FUNCTION_BLOCK FB_Camera
VAR_INPUT
END_VAR
VAR_OUTPUT
END_VAR
VAR
	Trigger	AT %Q*			: BOOL;				// signal to take picture and analyze
	CameraData				: ST_CameraData;	// modbus camera data
	VisionStatus			: ARRAY[0..3] OF BYTE;// modbus camera status
	_tubeParameters			: ST_TubeParameters;
	_pass					: BOOL;
	_fail					: BOOL;
	_noDetect				: BOOL;
			
	_xPoints 				: ARRAY[1..GVL.NumberVisionPoints] OF LREAL;
	_yPoints 				: ARRAY[1..GVL.NumberVisionPoints] OF LREAL;
	_xEllipsePoints			: ARRAY[1..GVL.NumberEllipsePoints] OF LREAL;
	_yEllipsePoints			: ARRAY[1..GVL.NumberEllipsePoints] OF LREAL;
		
	_displayVisionPts		: ARRAY[1..2,1..GVL.NumberVisionPoints] OF LREAL;
	_displayEllipsePts		: ARRAY[1..2,1..GVL.NumberEllipsePoints] OF LREAL;
	_columnPeak				: LREAL;	// xPeak value of the vision points
	_rowPeak				: LREAL;	// yPeak value of the vision points
	_rowCenterLine			: LREAL;	// based on entered minor value -> y value at the center-line axis
	_minorCalculated 		: LREAL;
	_majorCalculated		: LREAL;
	_xEllipseCenter			: LREAL;
	_yEllipseCenter			: LREAL;

	(* for calculating the pitch *)	
	_patternX1				: LREAL;
	_patternX2				: LREAL;
	_patternX3				: LREAL;
	_patternY1				: LREAL;
	_patternY2				: LREAL;
	_patternY3				: LREAL;
	
	(* calculation variables *)
	DeltaXpx				: LREAL;	// distance from peak of curve to center of cut (row)
	DeltaYpx				: LREAL;	// distance from peak of curve to center of cut (column)
	CutLength				: LREAL;
	CutHeight				: LREAL;
	DeltaXmm				: LREAL;
	DeltaYmm				: LREAL;
	(* results *)
	_CutLengthWithOffset	: LREAL;
	_DeltaXmmWithOffset		: LREAL;
	_DeltaYmmWithOffset		: LREAL;
	
	_depthOffset			: REAL; 				// difference due to the plane of cut is different than plane of pattern detect
	_minorRadiusMm			: LREAL := 2.5955;		// minor radius of ellipse in mm
	_majorRadiusMm			: LREAL;
	_slitCenterApparentRow	: LREAL;				// [px] this is the center of the part in x when accounting for the offset due to vision plane versus cut plane
	_tubeCenter				: LREAL;
	_tubeCenterOffset		: LREAL;
	_tubeCenterWithOffset	: LREAL;
	_cameraProgram			: STRING;
	_previousTubeIndex		: INT;
	
	_hmiParameters			: ST_CameraParameters;
	_parameters				: ST_CameraParameters;
	fbMessageChange			: FB_TcMessage;
	fbMessageLoaded			: FB_TcMessage;
END_VAR

PROPERTY angle : LREAL
GET
angle := _parameters.angle;
END_GET
SET
fbMessageChange.ipArguments.Clear().AddString('Angle').AddLReal(_parameters.angle).AddLReal(angle);
fbMessageChange.Send(0);
_parameters.angle := angle;
END_SET
END_PROPERTY

METHOD Calibrate : BOOL
VAR_INPUT
END_VAR
_hmiParameters.pitchRow := (CalibrationDistance / ABS(PatternY1 - PatternY2));
_hmiParameters.pitchColumn := (CalibrationDistance / ABS(PatternX2 - PatternX3));
END_METHOD

PROPERTY CalibrationDistance : LREAL
GET
CalibrationDistance := _parameters.calibrationDistance;
END_GET
SET
fbMessageChange.ipArguments.Clear().AddString('Calibration Distance').AddLReal(_parameters.calibrationDistance).AddLReal(CalibrationDistance);
fbMessageChange.Send(0);
_parameters.calibrationDistance := CalibrationDistance;
END_SET
END_PROPERTY

PROPERTY CameraProgram : STRING
GET
CameraProgram := _cameraProgram;
END_GET
SET
_cameraProgram := CameraProgram;
END_SET
END_PROPERTY

METHOD Compute : INT
VAR_INPUT
	Execute		: BOOL;
END_VAR
VAR_INST
	rTrig			: R_TRIG;
	nIndex			: INT;
	fbSecond		: FB_SecondOrder;
 	fbFourth		: FB_FourthOrder;
	fbEllipse		: FB_Ellipse;
	zeroValues		: BOOL;
END_VAR

VAR
	i: INT;
	yValue	: LREAL;
END_VAR
(* when computing the new cut positions, subtract the delta values from the 
original cut positions *)

rTrig(CLK := Execute);
IF rTrig.Q THEN
	nIndex := 10;
END_IF

IF NOT Execute THEN
	nIndex := 0;
END_IF

CASE nIndex OF
	0: // idle state
		Compute := 0;
	10: // get data
		IF GetCameraData() = 1 THEN
			nIndex := 15;
		END_IF
	15: // did pattern match find _xPoints, _yPoints?
		zeroValues := FALSE;
		FOR i := 1 TO GVL.NumberVisionPoints DO
			IF _xPoints[i] = 0 OR _yPoints[i] = 0 THEN
				zeroValues := TRUE;
			END_IF
		END_FOR
		IF zeroValues THEN
			nIndex := 60;
		ELSE
			nIndex := 20;
		END_IF
	20: // compute the peak x value of the data		
		fbSecond.FindPeak(xValues := ADR(_xPoints), yValues := ADR(_yPoints), xPeak := ADR(_columnPeak));
		fbFourth.FindYatX(xValues := ADR(_xPoints), yValues := ADR(_yPoints), xPeak := ADR(_columnPeak), yPeak := ADR(_rowPeak));
		DeltaYpx := CameraData.Results.LocationInX - _columnPeak;
		DeltaYmm := DeltaYpx * _hmiParameters.pitchColumn;
		_DeltaYmmWithOffset := DeltaYmm + _tubeParameters.AdjustmentY;
		
		CutLength := CameraData.Results.WidthMeasurement * _hmiParameters.pitchColumn;		
		_CutLengthWithOffset := CutLength + _tubeParameters.AdjustmentLength;
		CutHeight := CameraData.Results.HeightMeasurement * _hmiParameters.pitchRow;
		
		_tubeCenter := _rowPeak + 0.5*_tubeParameters.Diameter /_hmiParameters.pitchRow;
		_tubeCenterOffset := (_tubeParameters.DepthOfPocket*TAN(_hmiParameters.angle * 2*3.14159/360.0))/_hmiParameters.pitchRow;
		_tubeCenterWithOffset := _tubeCenter + _tubeCenterOffset;
		
		DeltaXpx := (CameraData.Results.LocationInY - 0.5*CameraData.Results.HeightMeasurement) - _tubeCenterWithOffset;
		DeltaXmm := DeltaXpx * _hmiParameters.pitchRow;
		_DeltaXmmWithOffset := DeltaXmm + _tubeParameters.AdjustmentX;
		
		nIndex := 50;
	30: // compute ellipse
		fbEllipse.EllipseFit(xValues := _xEllipsePoints, yValues := _yEllipsePoints);
		nIndex := 40;
		
	40: // assign values
		_minorCalculated := fbEllipse.minor;
		_majorCalculated := fbEllipse.major;
		_xEllipseCenter := fbEllipse.centrex;
		_yEllipseCenter := fbEllipse.centrey;
		nIndex := 50;
	50: // done state
		Compute := 1;		
	60: // didn't find the pattern, so can't compute a peak
		Compute := -1;					
END_CASE
END_METHOD

PROPERTY CutLengthWithOffset : LREAL
GET
CutLengthWithOffset := _CutLengthWithOffset;
END_GET
END_PROPERTY

PROPERTY DeltaXmmWithOffset : LREAL
GET
DeltaXmmWithOffset := _DeltaXmmWithOffset;
END_GET
END_PROPERTY

PROPERTY DeltaYmmWithOffset : LREAL
GET
DeltaYmmWithOffset := _DeltaYmmWithOffset;
END_GET
END_PROPERTY

PROPERTY Fail : BOOL
GET
Fail := _fail;
END_GET
SET
_fail := Fail;
END_SET
END_PROPERTY

METHOD FB_init : BOOL
VAR_INPUT
	bInitRetains : BOOL; // if TRUE, the retain variables are initialized (warm start / cold start)
	bInCopyCode : BOOL;  // if TRUE, the instance afterwards gets moved into the copy code (online change)
END_VAR
IF NOT fbMessageChange.EqualsToEventEntryEx(stOther := TC_EVENTS.SlitterEvents.ParameterChange) THEN
	fbMessageChange.CreateEx(TC_EVENTS.SlitterEvents.ParameterChange, 0);
	fbMessageChange.ipArguments.Clear();
END_IF

IF NOT fbMessageLoaded.EqualsToEventEntryEx(stOther := TC_EVENTS.SlitterEvents.ParametersLoadedFromFile) THEN
	fbMessageLoaded.CreateEx(TC_EVENTS.SlitterEvents.ParametersLoadedFromFile, 0);
	fbMessageLoaded.ipArguments.Clear().AddString('Camera');
END_IF
END_METHOD

METHOD GetCameraData : INT
VAR_INPUT
END_VAR

VAR_INST
	i				: INT;
	fbMBRegRead		: FB_MBReadRegs;
END_VAR
// format on Cognex needs to be little endian 
GetCameraData := 0;
fbMBRegRead.bExecute := TRUE;

fbMBRegRead.sIPAddr := GVL.CameraIpAddress;
fbMBRegRead.nTCPPort := 502;
fbMBRegRead.nUnitID := 16#FF;
fbMBRegRead.nQuantity := 94; // 188/2;
fbMBRegRead.nMBAddr := GVL.ModbusReadOffset+5;
fbMBRegRead.cbLength := SIZEOF(CameraData.Results);
fbMBRegRead.pDestAddr := ADR(CameraData.Results);

fbMBRegRead();

IF NOT fbMBRegRead.bBusy THEN
	IF NOT fbMBRegRead.bError THEN
		fbMBRegRead(bExecute := FALSE);
		FOR i := 1 TO GVL.NumberVisionPoints DO
			_yPoints[i] := REAL_TO_LREAL(CameraData.Results.PointValueRow[i]);
			_xPoints[i] := REAL_TO_LREAL(CameraData.Results.PointValueColumn[i]);
			_displayVisionPts[1,i] := INT_TO_LREAL(LREAL_TO_INT(_xPoints[i]*100))/100.0; // column values
			_displayVisionPts[2,i] := INT_TO_LREAL(LREAL_TO_INT(_yPoints[i]*100))/100.0; // row values	
		END_FOR

		GetCameraData := 1;	
	ELSE
		fbMBRegRead(bExecute := FALSE);
		FOR i := 1 TO GVL.NumberVisionPoints DO
			_xPoints[i] := 0;
			_yPoints[i] := 0;
			_displayVisionPts[1,i] := 0;
			_displayVisionPts[2,i] := 0;
	
		END_FOR
		GetCameraData := -1;	
		
	END_IF
END_IF
END_METHOD

METHOD Inspect : INT
VAR_INPUT
	Execute	: BOOL;
END_VAR
VAR_INST
	nIndex 	: INT;
	rTrig	: R_TRIG;
	CountStart : REAL;
	CountFinish : REAL;
	Count	: REAL;
	CameraTON	: TON := (PT := T#250MS);
	CameraDataResult : INT;
END_VAR
rTrig(CLK := Execute);
IF rTrig.Q THEN
	Inspect := 0;
	nIndex := 10;
	Trigger := FALSE;
	Compute(Execute := FALSE);
	CameraTON(IN := FALSE);
END_IF

IF NOT Execute THEN
	nIndex := 0;
END_IF

CASE nIndex OF
	0: // idle state
		Inspect := 0;
	10: // trigger the camera
		IF GetCameraData() = 1 THEN
			Count := CameraData.Results.Count;
			CountStart := CameraData.Results.Count;
			nIndex := 11;
		END_IF
	11: // trigger camera
		Trigger := TRUE;
		nIndex := 12;
	12: // wait 250 ms
		CameraTON.IN := TRUE;
		IF CameraTON.Q THEN
			CameraTON.IN := FALSE;
			nIndex := 15;
		END_IF
		CameraTON();
	15: // wait for data to be updated
		CameraDataResult := GetCameraData();
		IF CameraDataResult = 1 THEN
			IF Count <> CameraData.Results.Count THEN
				CountFinish := CameraData.Results.Count;
				nIndex := 20;
				Trigger := FALSE;
			END_IF
		END_IF
	20: // Gather the data and analyze locations, etc.
		CameraDataResult := Compute(Execute := TRUE);
		IF CameraDataResult = 1 THEN	// could compute b/c found pattern
			Compute(Execute := FALSE);
			nIndex := 30;	
		ELSIF CameraDataResult = -1 THEN	// could not comput b/c no pattern found
			Compute(Execute := FALSE);
			nIndex := 50;
		END_IF
	30: // compute pass fail
		IF PassFail() THEN	// true = pass
			_pass := TRUE;
			_fail := FALSE;
			_noDetect := FALSE;
		ELSE
			_pass := FALSE;
			_fail := TRUE;
			_noDetect := FALSE;
		END_IF
		nIndex := 40;
	40: // done state
		Inspect := 1;
	50: // error state
		Inspect := -1;
		_noDetect := TRUE;		
		_pass := FALSE;
		_fail := FALSE;		
END_CASE
END_METHOD

METHOD MonitorParameters : BOOL
VAR_INPUT
END_VAR
IF angle <> _hmiParameters.angle THEN
	angle := _hmiParameters.angle;
END_IF

IF CalibrationDistance <> _hmiParameters.calibrationDistance THEN
	CalibrationDistance := _hmiParameters.calibrationDistance;
END_IF

IF pitchColumn <> _hmiParameters.pitchColumn THEN
	pitchColumn := _hmiParameters.pitchColumn;
END_IF

IF pitchRow <> _hmiParameters.pitchRow THEN
	pitchRow := _hmiParameters.pitchRow;
END_IF
END_METHOD

PROPERTY NoDetect : BOOL
GET
NoDetect := _noDetect;
END_GET
SET
_noDetect := NoDetect;
END_SET
END_PROPERTY

PROPERTY Parameters : ST_CameraParameters
GET
Parameters := _parameters;
END_GET
SET
_parameters := Parameters;
_hmiParameters := Parameters;
fbMessageLoaded.Send(0);
END_SET
END_PROPERTY

PROPERTY Pass : BOOL
GET
Pass := _pass;
END_GET
SET
_pass := Pass;
END_SET
END_PROPERTY

METHOD PassFail : BOOL
VAR_INPUT
END_VAR
PassFail := TRUE; // set to pass and overwrite if anything causes failure;

// cut length
IF _tubeParameters.AdjustmentLength + CutLength > _tubeParameters.MaxLength OR
	_tubeParameters.AdjustmentLength + CutLength < _tubeParameters.MinLength THEN
		PassFail := FALSE;
END_IF

// delta x
IF ABS(_tubeParameters.AdjustmentX + DeltaXmm) > _tubeParameters.ResultToleranceX THEN
	PassFail := FALSE;
END_IF

// delta y
IF ABS(_tubeParameters.AdjustmentY + DeltaYmm) > _tubeParameters.ResultToleranceY THEN
	PassFail := FALSE;
END_IF

// height
IF CutHeight < _tubeParameters.MinHeight OR CutHeight > _tubeParameters.MaxHeight THEN
	PassFail := FALSE;
END_IF
END_METHOD

PROPERTY PatternMatchX : LREAL
GET
PatternMatchX := REAL_TO_LREAL(CameraData.Results.PatternMatchColumn);
END_GET
END_PROPERTY

PROPERTY PatternMatchY : LREAL
GET
PatternMatchY := REAL_TO_LREAL(CameraData.Results.PatternMatchRow);
END_GET
END_PROPERTY

PROPERTY PatternX1 : LREAL
GET
PatternX1 := _patternX1;
END_GET
SET
_patternX1 := PatternX1;
END_SET
END_PROPERTY

PROPERTY PatternX2 : LREAL
GET
PatternX2 := _patternX2;
END_GET
SET
_patternX2 := PatternX2;
END_SET
END_PROPERTY

PROPERTY PatternX3 : LREAL
GET
PatternX3 := _patternX3;
END_GET
SET
_patternX3 := PatternX3;
END_SET
END_PROPERTY

PROPERTY PatternY1 : LREAL
GET
PatternY1 := _patternY1;
END_GET
SET
_patternY1 := PatternY1;
END_SET
END_PROPERTY

PROPERTY PatternY2 : LREAL
GET
PatternY2 := _patternY2;
END_GET
SET
_patternY2 := PatternY2;
END_SET
END_PROPERTY

PROPERTY PatternY3 : LREAL
GET
PatternY3 := _patternY3;
END_GET
SET
_patternY3 := PatternY3;
END_SET
END_PROPERTY

PROPERTY pitchColumn : LREAL
GET
pitchColumn := _parameters.pitchColumn;
END_GET
SET
fbMessageChange.ipArguments.Clear().AddString('pitchColumn').AddLReal(_parameters.pitchColumn).AddLReal(pitchColumn);
fbMessageChange.Send(0);
_parameters.pitchColumn := pitchColumn;
END_SET
END_PROPERTY

PROPERTY PitchMmToPixel : LREAL
GET
PitchMmToPixel := _hmiParameters.pitchRow;
END_GET
END_PROPERTY

PROPERTY pitchRow : LREAL
GET
pitchRow := _parameters.pitchRow;
END_GET
SET
fbMessageChange.ipArguments.Clear().AddString('pitchRow').AddLReal(_parameters.pitchRow).AddLReal(pitchRow);
fbMessageChange.Send(0);
_parameters.pitchRow := pitchRow;
END_SET
END_PROPERTY

METHOD SelectCameraProgram : INT
VAR_INPUT
	Execute	: BOOL;
END_VAR
VAR_INST
	fbMBRegWrite 	: FB_MBWriteRegs;	// for writing command, name; offset is 2000
	fbMBCoilWrite	: FB_MBWriteCoils;	// for writing vision control; offset is 0
	fbMBReadInputs 	: FB_MBReadInputs; 	// for reading vision status; offset is 0
	nIndex			: INT;
	rTrig			: R_TRIG;
	JobLoadByName 	: WORD := 16#4000;
	temp 			: UDINT := 0;
	info 			: BOOL;
	i 				: WORD;
	strJobName 		: STRING;
	Message			: STRING(255);
	ErrorId			: UDINT;
	nQuantity 		: WORD;
	cbLength 		: UDINT;	
	attempt			: INT;
	attempt2		: INT;	
END_VAR
VAR
END_VAR
rTrig(CLK := Execute);
IF rTrig.Q THEN
	nIndex := 10;
	Message := '';
	ErrorId := 0;
	Attempt := 0;
	Attempt2 := 0;
	fbMBCoilWrite(
		bExecute := FALSE,
		sIPAddr := GVL.CameraIpAddress,
		nTCPPort := 502,
		nUnitID := 16#FF);
	fbMBRegWrite(
		bExecute := FALSE,
		sIPAddr := GVL.CameraIpAddress,
		nTCPPort := 502,
		nUnitID := 16#FF);
	fbMBReadInputs(
		bExecute := FALSE,
		sIPAddr := GVL.CameraIpAddress,
		nTCPPort := 502,
		nUnitID := 16#FF);
END_IF

IF NOT Execute THEN
	nIndex := 0;
END_IF

CASE nIndex OF
	0: // idle state
		SelectCameraProgram := 0;
	10: // check if the program needs to change
		IF _previousTubeIndex = _tubeParameters.Index THEN
			nIndex := 75;
		ELSE
			nIndex := 15;
		END_IF
	15: // Reset everything to zero
		fbMBCoilWrite(
			nQuantity := 32,
			nMBAddr := 0,
			cbLength := 4,
			pSrcAddr := ADR(temp),
			bExecute := TRUE);
		IF NOT fbMBCoilWrite.bBusy THEN
			fbMBCoilWrite(bExecute := FALSE);
			nIndex := 20;
		END_IF
		IF fbMBCoilWrite.bError THEN
			Message := 'Error in state 15';
			ErrorId := fbMBCoilWrite.nErrId;
			fbMBCoilWrite(bExecute := FALSE);
			nIndex := 85;
		END_IF
	20: // place camera offline by setting the set offline bit high 
		// modbus coil offset is 0
		// byte 0, bit 7 is the bit for forcing the camera to be offline
		info := TRUE;
		fbMBCoilWrite(
			sIPAddr := GVL.CameraIpAddress,
			nTCPPort := 502,
			nUnitID := 16#FF,
			nQuantity := 1,
			nMBAddr := 7,
			cbLength := 1,
			pSrcAddr := ADR(Info),
			bExecute := TRUE);
		IF NOT fbMBCoilWrite.bBusy THEN
			fbMBCoilWrite(bExecute := FALSE);
			nIndex := 30;
			END_IF
		IF fbMBCoilWrite.bError THEN
			Message := 'Error in state 20';
			ErrorId := fbMBCoilWrite.nErrId;
			fbMBCoilWrite(bExecute := FALSE);
			nIndex := 85;
		END_IF		
	30: // write the job load by name command into Word 0 of the input block 
		// job load by name command is 0x4000
		// this goes into holding register start which is at 2000
		fbMBRegWrite(
			nQuantity := 1,
			nMBAddr := GVL.ModbusWriteOffset,
			cbLength := 2,
			pSrcAddr := ADR(JobLoadByName),
			bExecute := TRUE);
		IF NOT fbMBRegWrite.bBusy THEN
			fbMBRegWrite(bExecute := FALSE);
			attempt := attempt + 1;
			IF attempt > 2 THEN
				attempt := 0;
				nIndex := 40;
			END_IF
		END_IF
		IF fbMBRegWrite.bError THEN
			Message := 'Error in state 30';
			ErrorId := fbMBRegWrite.nErrId;
			fbMBRegWrite(bExecute := FALSE);
			nIndex := 85;

		END_IF
	40: // write the job name to Word 1 - 2000 (UserData).  Job name must be null terminated
		// a 0 must be in the byte immediately following the job name
		strJobName := CONCAT('SDCARD/Tube', INT_TO_STRING(_tubeParameters.Index));
		strJobName := CONCAT(strJobName, '.job');
		cbLength := 18; // INT_TO_UDINT(LEN(strJobName) + 1);
		nQuantity := 9; //REAL_TO_WORD(UDINT_TO_REAL(cbLength)/2);
		fbMBRegWrite(
			bExecute := TRUE,
			nQuantity := nQuantity,
			nMBAddr := GVL.ModbusWriteOffset + 1,
	//		nQuantity := nQuantity, // number of words
			cbLength := cbLength, // byte size
			pSrcAddr := ADR(strJobName));
		IF NOT fbMBRegWrite.bBusy THEN
			fbMBRegWrite(bExecute := FALSE);
			nIndex := 50;
		END_IF			
		IF fbMBRegWrite.bError THEN
			Message := 'Error in state 40';
			ErrorId := fbMBRegWrite.nErrId;
			fbMBRegWrite(bExecute := FALSE);
			Attempt2 := Attempt2 + 1;
			IF attempt2 > 2 THEN
				nIndex := 85;
			END_IF
		END_IF
		
	50: // Set the Execute Command bit in the vision control block
		//VisionControl.ExecuteCommand := TRUE;
		// Byte 0, bit 4 of vision control 
		info := TRUE;
		fbMBCoilWrite(
			nQuantity := 1,
			nMBAddr := 4,
			cbLength := 1,
			pSrcAddr := ADR(Info),
			bExecute := TRUE);
		IF NOT fbMBCoilWrite.bBusy THEN
			fbMBCoilWrite(bExecute := FALSE);
			nIndex := 60;
		END_IF
		IF fbMBCoilWrite.bError	THEN
			fbMBCoilWrite(bExecute := FALSE);
			nIndex := 85;
			Message := 'error in state 50';
			errorid := fbMBCoilWrite.nErrId;
		END_IF
	60: // wait for command complete of command failed to be set before clearing the execute
		// command bit and the offline bit
		fbMBReadInputs(
			sIPAddr := GVL.CameraIpAddress,
			nTCPPort := 502,
			nUnitID := 16#FF,
			nQuantity := 32,
			nMBAddr := 0,
			cbLength := 4,
			pDestAddr := ADR(VisionStatus),
			bExecute := TRUE);
		IF NOT fbMBReadInputs.bBusy THEN
			fbMBReadInputs(bExecute := FALSE);
			IF VisionStatus[1].6 OR VisionStatus[1].5 THEN
				nIndex := 70;
				IF VisionStatus[1].6 THEN
					nIndex := 80;
					Message := 'VisionSatus[1].6 is true.';
				END_IF
			END_IF
		END_IF
		IF fbMBReadInputs.bError THEN
			fbMBReadInputs(bExecute := FALSE);
			nIndex := 85;
			Errorid := fbMBReadInputs.nErrId;
			Message := 'errror in state 60.';
		END_IF
	70: // done state
		fbMBCoilWrite(
			nQuantity := 32,
			nMBAddr := 0,
			cbLength := 4,
			pSrcAddr := ADR(temp),
			bExecute := TRUE);
		IF NOT fbMBCoilWrite.bBusy THEN
			fbMBCoilWrite(bExecute := FALSE);
			nIndex := 75;
		END_IF
		IF fbMBCoilWrite.bError THEN
			fbMBCoilWrite(bExecute := FALSE);
			nIndex := 85;
			Message := 'error in state 70';
			ErrorID := fbMBCoilWrite.nErrId;			
		END_IF
	75: // done state
		_previousTubeIndex := _tubeParameters.Index;
		SelectCameraProgram := 1;
	80: // error state
		fbMBCoilWrite(
			nQuantity := 32,
			nMBAddr := 0,
			cbLength := 4,
			pSrcAddr := ADR(temp),
			bExecute := TRUE);
		IF NOT fbMBCoilWrite.bBusy THEN
			fbMBCoilWrite(bExecute := FALSE);
			nIndex := 85;
		END_IF

	85: // error state
		SelectCameraProgram := -1;
END_CASE





(*
SelectCameraProgram := 0;
fbMBRegWrite.bExecute := TRUE;

fbMBRegWrite.sIPAddr := GVL.CameraIpAddress;
fbMBRegWrite.nTCPPort := 502;
fbMBRegWrite.nUnitID := 16#FF;
fbMBRegWrite.nQuantity := 2; // words to write
fbMBRegWrite.nMBAddr := GVL.ModbusWriteOffset;
fbMBRegWrite.cbLength := SIZEOF(_tubeSelection);
fbMBRegWrite.pSrcAddr := ADR(_tubeSelection);

fbMBRegWrite();

IF NOT fbMBRegWrite.bBusy THEN
	IF NOT fbMBRegWrite.bError THEN
		fbMBRegWrite(bExecute := FALSE);
		SelectCameraProgram := 1;
	ELSE
		fbMBRegWrite(bExecute := FALSE);
		SelectCameraProgram := -1;		
	END_IF
END_IF
*)
END_METHOD

METHOD TriggerCamera : BOOL
VAR_INPUT
	Execute	: BOOL;
END_VAR
VAR_INST
	rTrig	: R_TRIG;
	nIndex	: INT;
	Counter	: REAL;
END_VAR
rTrig(CLK := Execute);
IF rTrig.Q THEN
	nIndex := 10;
	Trigger	:= FALSE;
END_IF

IF NOT Execute THEN
	nIndex := 0;
END_IF

CASE nIndex OF
	0: // idle state
		TriggerCamera := FALSE;
	10: // get the camera count
		IF GetCameraData() = 1 THEN
			Counter := CameraData.Results.Count;
			nIndex := 20;
		END_IF
	20: // trigger the camera	
		Trigger := TRUE;
		IF GetCameraData() = 1 THEN
			nIndex := 30;
		END_IF
	30: // updated?
		IF Counter <> CameraData.Results.Count THEN
			Trigger := FALSE;
			nIndex := 40;
		ELSE
			nIndex := 20;
		END_IF
	40: // done state
		TriggerCamera := TRUE;
END_CASE
END_METHOD

PROPERTY TubeParameters : ST_TubeParameters
GET
TubeParameters := _tubeParameters;
END_GET
SET
_tubeParameters := TubeParameters;
END_SET
END_PROPERTY

PROPERTY xEllipseCenter : LREAL
GET
xEllipseCenter := _xEllipseCenter;
END_GET
END_PROPERTY

PROPERTY yEllipseCenter : LREAL
GET
yEllipseCenter := _yEllipseCenter;
END_GET
END_PROPERTY

END_FUNCTION_BLOCK

(* stored: Version 1.1.0.1, ProductVersion 3.1.4024.9
   POU FB_Camera: Id {e29b8acf-c363-459e-aac4-9b2f4b8da33e}, SpecialFunc None
   Folder Parameters: Id {c3f8c6ab-b4bb-432d-94e3-1b6e85c8648c}
   Property angle: Id {9837e397-79d0-4c7d-9c41-c597cf42d2a2}
   Get Get: Id {8d796e00-e9a8-41d8-aa78-baf730d2028b}
   Set Set: Id {ccf7781c-4d23-4e7d-a804-57aafb8844c9}
   Method Calibrate: Id {47bb793d-9a4a-46a0-8f3e-b2726fff7b46}
   Property CalibrationDistance: Id {d5b16c9d-22ca-470b-9a6e-4cd0a967eaf7}
   Get Get: Id {4f7a49bd-d4f7-4486-8398-861beff2278d}
   Set Set: Id {77981a05-efbd-441b-9460-6e5d2f43a673}
   Property CameraProgram: Id {fd3b28ca-4e8a-47f7-8989-29a9cd3cb0b3}
   Get Get: Id {e3b7765f-f4a0-4831-8af9-5860050b203d}
   Set Set: Id {35833dfc-12e1-42b2-8f0f-62d8d96f08ba}
   Method Compute: Id {317c842b-2189-4bec-b370-314b3f33f4a1}
   Property CutLengthWithOffset: Id {b454241c-1d74-4f31-a305-41796035a30d}
   Get Get: Id {28adb857-d7ba-41a8-9a50-8a94af4a60a3}
   Property DeltaXmmWithOffset: Id {a355d9c0-b275-4ede-94bc-4d7ced197860}
   Get Get: Id {0b155c76-beb9-496c-9de0-09505182dbfa}
   Property DeltaYmmWithOffset: Id {1638acf8-e7a1-4300-b8d2-17caa2f29476}
   Get Get: Id {1a4f4740-3f40-4eef-945b-008971e7f564}
   Property Fail: Id {00e3ce85-e94d-4899-a632-72a1ffd4c881}
   Get Get: Id {5440d75f-b626-49d3-92f7-2739997c7a0b}
   Set Set: Id {106c6fe7-b712-467c-bb5a-172fb08dea35}
   Method FB_init: Id {9bcee5cd-fdb6-467b-a10e-19b74865c7d4}
   Method GetCameraData: Id {196673c8-e986-4d26-9da6-677accad1607}
   Method Inspect: Id {afb340ef-d650-47e6-aff6-56214386a178}
   Method MonitorParameters: Id {8de04281-1ba7-4484-b717-19caaf5ae689}
   Property NoDetect: Id {20e83035-70d3-4a21-9b8e-71e1ba4c26ab}
   Get Get: Id {44d3ded5-83e8-40c5-a078-604500e88c36}
   Set Set: Id {7d900a17-473a-467b-afa0-dc329071e819}
   Property Parameters: Id {0a912b95-5702-423f-ad14-f73625868c44}
   Get Get: Id {9004d6db-23fd-4a0e-acca-0c657f2ab045}
   Set Set: Id {0c0dd0c0-9c65-4816-83c9-62c59ac11cf5}
   Property Pass: Id {e23aae12-0dd3-45cb-8509-aca8f81a2b79}
   Get Get: Id {5c452049-6ba1-48a5-afec-c835cf5432b7}
   Set Set: Id {42838619-486c-482b-ae24-9fe96a670a6b}
   Method PassFail: Id {fd5bc711-f02b-40fe-bb25-b8c1462f30e0}
   Property PatternMatchX: Id {e856e423-371b-459d-96cd-c9c3a9871218}
   Get Get: Id {db3578a3-2e6c-4db5-b9ea-da8eaa4b62e5}
   Property PatternMatchY: Id {f794541b-d0f4-43f5-9989-f5b72f46a724}
   Get Get: Id {afe4b227-5eb1-4637-8576-982aaa1d7cee}
   Property PatternX1: Id {34a1f4f2-d6c3-40ba-a56f-6e8bac116405}
   Get Get: Id {aca48926-3280-4f5d-9704-de65a56549f7}
   Set Set: Id {71d553df-b96f-404c-adc2-a73157f57b7a}
   Property PatternX2: Id {f6e6ef21-611a-49fd-b20d-6fa0e51ee685}
   Get Get: Id {ceb1abeb-4be0-4990-ab6b-2bb8e6d573f9}
   Set Set: Id {06302c94-72d4-4a46-8071-c1d6c8020f7f}
   Property PatternX3: Id {3f489872-a246-4f21-8a7b-d024b4b714c3}
   Get Get: Id {5d750c6a-9c90-4cd6-b09d-26abb56916fa}
   Set Set: Id {72d5c483-34b4-4d23-9625-06173b7466de}
   Property PatternY1: Id {0625def3-faa7-4cce-961b-14de7462443d}
   Get Get: Id {51ba8222-4e92-47bc-a423-7b36abb6dc7f}
   Set Set: Id {8a6a9157-340a-46de-9ae8-8d516456b3c6}
   Property PatternY2: Id {bac46706-290a-454b-b2b6-45489dbfb721}
   Get Get: Id {93812042-9add-4a65-8b67-67111a707288}
   Set Set: Id {30a03a69-0055-406a-a28e-0a5368bf59ba}
   Property PatternY3: Id {2994abb7-2d25-4e87-a172-de7ded7dd3ba}
   Get Get: Id {89b27ac1-e922-43f4-a5d0-4ea216603666}
   Set Set: Id {b4e772fc-cc30-4535-b999-b96bc0cf7943}
   Property pitchColumn: Id {9a251985-6952-4587-8a62-c2789e7fe16a}
   Get Get: Id {9a70de58-d5e8-4958-8a9f-5bd64f861a81}
   Set Set: Id {e881a551-ee32-4f57-b2cf-a73f32117acd}
   Property PitchMmToPixel: Id {fb91ea54-ce4d-40c4-af64-be5e57a50eb3}
   Get Get: Id {c424417a-2fa7-4a18-ab34-5982a15bc656}
   Property pitchRow: Id {035ad7e2-9f28-41de-8283-767f0518893e}
   Get Get: Id {5ba2f54a-a285-4cef-853a-57bbf819858f}
   Set Set: Id {d9843d7d-e848-4635-91ec-9b88afcf8a15}
   Method SelectCameraProgram: Id {00e1d34d-f3f7-42d4-99f2-f1957dfadecb}
   Method TriggerCamera: Id {9239a2ac-48e0-4f63-b1b4-182558d5e90b}
   Property TubeParameters: Id {400ab4f1-96e8-4818-a86c-ef0f62c8cde6}
   Get Get: Id {5df344ac-de22-402d-9618-4c0f5046ddaf}
   Set Set: Id {b5d2b68a-f3e6-45a3-bebc-0314a00bb16a}
   Property xEllipseCenter: Id {86f1bf78-74fd-43c9-9b64-b7e7835b5035}
   Get Get: Id {839c6b74-3a8b-4dab-8bc3-0baf0a96597f}
   Property yEllipseCenter: Id {bc3ea8e2-c6ec-4170-acbe-bd54fe16cf38}
   Get Get: Id {2d0da89b-5f70-401e-b43d-d9ca521ee0ea} *)
